Universal Robots URScript: movej_example2.script

def movej_example2():

  set_standard_analog_input_domain(0, 1)
  set_standard_analog_input_domain(1, 1)
  set_tool_analog_input_domain(0, 1)
  set_tool_analog_input_domain(1, 1)
  set_analog_outputdomain(0, 0)
  set_analog_outputdomain(1, 0)
  set_tool_voltage(0)
  set_input_actions_to_default()
  set_tcp(p[0.0,0.0,0.0,0.0,0.0,0.0])
  set_payload(0.0)
  set_gravity([0.0, 0.0, 9.82])
  global Point_1=p[0.20357790895191322,-0.2889867422664357,0.5839434681846556,0.8910156392575451,1.0478765804907595,0.9454746698760753]

  q1 = [-4.3582165175113925, -1.5556169457521332, 1.5001790238252788, -0.2975105484571863, 0.8263615579881575, -0.06287913030982217]
  q2 = [-3.9459161143182633, -1.5804172826659855, 1.8665460616996652, -0.6273449535274391, 0.8628807654549796, -0.08054465460352489]
  q3 = [-3.329116114318263, -1.5804172826659855, 1.8665460616996652, -0.6273449535274391, 0.8628807654549796, -0.08054465460352489]

  a_q = 1.3962634015954636
  v_q = 1.0471975511965976

  pose1 = [-2.6563161143182623, -1.3393135326659849, 1.8665460616996652, -0.6273449535274391, 0.8628807654549796, -0.08054465460352489]
  pose2 = [-2.65631611441043, -1.4664110736586835, 1.4816798984770223, -0.11538124931998528, 0.8628807653632613, -0.08054465459140303]

  a_p = 1.2
  v_p = 0.25

  while (True):
    movej(q1, a_q, v_q)

    movej(q2, a_q, v_q)

    movej(q3, a_q, v_q)


    movel(pose1, a_p, v_p)

    movel(pose2, a_p, v_p)
  end

end
